{attribute 'GeneratedUsingTerminal: EL1052-0000-0016'}
{attribute addProperty BoxType "EL1052-0000-0016"}
{attribute addProperty Id "InputAT %I*BOOL1ErrorAT %I*BOOL1"}
{attribute addProperty CRC "835648127"}
{attribute addProperty Size "2"}
TYPE Channel_31CEFA7F :
STRUCT
	{attribute addProperty Name "Input"}
	Input AT %I* : BOOL;
	{attribute addProperty Name "Error"}
	Error AT %I* : BOOL;
END_STRUCT
END_TYPE

(* stored: Version 1.2.0.0, ProductVersion 3.1.4024.9
   DUT Channel_31CEFA7F: Id {a884c84b-74b5-4dbd-bb13-d78a01255264} *)
